// TwinCAT 3 PLC project plc_eta_factory_climate_room_automation
// ProgramVersion: 3.1.4024.12
// libraries:
//   AutomationBaseClasses, * (PTW TU Darmstadt)
//   Tc2_ControllerToolbox, * (Beckhoff Automation GmbH)
//   Tc2_MBus, * (Beckhoff Automation GmbH)
//   Tc2_Standard, * (Beckhoff Automation GmbH)
//   Tc2_System, * (Beckhoff Automation GmbH)
//   Tc2_Utilities, * (Beckhoff Automation GmbH)
//   Tc3_Module, * (Beckhoff Automation GmbH)
// project tree:
//   DUTs/04 Systems/ E_ActiveWallModulesControlMode.TcDUT, E_AirHandlingUnitControlMode.TcDUT, ST_ActiveWallModulesDefaultParameters.TcDUT, ST_ActiveWallModulesSetParameters.TcDUT, ST_AirHandlingUnitDefaultParameters.TcDUT, ST_PowerControlledHeaterState.TcDUT, ST_PowerControlledHeaterDefaultParameters.TcDUT, ST_AirHandlingUnitSetParameters.TcDUT, ST_AmbientState.TcDUT, ST_BufferStorageState.TcDUT
//   GVLs/ GlobalVariables.TcGVL, MBus.TcGVL
//   / MBusTask.TcTTO, PlcTask.TcTTO
//   POUs/01 Actuators/ FB_AirHandlingUnit.TcPOU, FB_PowerControlledHeaterThyristor.TcPOU, FB_PowerControlledHeaterFan.TcPOU, FB_PowerControlledHeaterContactor.TcPOU
//   POUs/02 Sensors/ FB_CO2Sensor.TcPOU, FB_HumiditySensor.TcPOU, FB_TemperatureSensor.TcPOU, FB_TemperatureSensorPCH.TcPOU, FB_JanitzaSensor.TcPOU
//   POUs/04 Systems/ FB_ActiveWallModulesSystem.TcPOU, FB_AirHandlingUnitSystem.TcPOU, FB_Ambient.TcPOU, FB_BufferStorage.TcPOU, FB_CNSystem.TcPOU, FB_HNLTSystem.TcPOU, FB_PowerControlledHeaterSystem.TcPOU
//   POUs/ MAIN.TcPOU, MBus_Communication.TcPOU

CONFIGURATION plc_eta_factory_climate_room_automation
    RESOURCE PLC ON TwinCAT3
        TASK MBusTask(INTERVAL := T#10ms, PRIORITY := 1);
        TASK PlcTask(INTERVAL := T#10ms, PRIORITY := 20);
        PROGRAM MBus_Communication WITH MBusTask : MBus_Communication;
        PROGRAM MAIN WITH PlcTask : MAIN;
    END_RESOURCE
END_CONFIGURATION

// ---- DUTs/04 Systems/E_ActiveWallModulesControlMode.TcDUT
{attribute 'qualified_only'}
{attribute 'strict'}
TYPE E_ActiveWallModulesControlMode :
(
	On := 0, //100% on
	Discrete := 1, //use hysteresis controller
	Continous := 2 //use PI-Controller
);
END_TYPE

// ---- DUTs/04 Systems/E_AirHandlingUnitControlMode.TcDUT
{attribute 'qualified_only'}
{attribute 'strict'}
TYPE E_AirHandlingUnitControlMode :
(
	On := 0, //100% on
	Discrete := 1, //use hysteresis controller
	Continous := 2 //use PI-Controller
);
END_TYPE

// ---- DUTs/04 Systems/ST_ActiveWallModulesDefaultParameters.TcDUT
TYPE ST_ActiveWallModulesDefaultParameters :
STRUCT
	aSetPointLimitsTemperature : ARRAY[1..2] OF REAL := [5,30];
END_STRUCT
END_TYPE

// ---- DUTs/04 Systems/ST_ActiveWallModulesSetParameters.TcDUT
{attribute 'OPC.UA.DA.StructuredType' := '1'}
TYPE ST_ActiveWallModulesSetParameters :
STRUCT
	bHeatingModeAlgorithm : BOOL;
	bHeatingModeManual : BOOL;
	nControlModeAlgorithm : E_ActiveWallModulesControlMode;
	nControlModeManual : E_ActiveWallModulesControlMode;
	fHysteresisRangeAlgorithm : REAL;
	fHysteresisRangeManual : REAL; 
END_STRUCT
END_TYPE

// ---- DUTs/04 Systems/ST_AirHandlingUnitDefaultParameters.TcDUT
TYPE ST_AirHandlingUnitDefaultParameters :
STRUCT
	aSetPointLimitsTemperature : ARRAY[1..2] OF REAL := [5,100];
END_STRUCT
END_TYPE

// ---- DUTs/04 Systems/ST_PowerControlledHeaterState.TcDUT
{attribute 'OPC.UA.DA.StructuredType' := '1'}
TYPE ST_PowerControlledHeaterState :
STRUCT
	fPowerTotal : REAL;
	sPowerUnit : STRING := 'W';
END_STRUCT
END_TYPE

// ---- DUTs/04 Systems/ST_PowerControlledHeaterDefaultParameters.TcDUT
TYPE ST_PowerControlledHeaterDefaultParameters :
STRUCT
	aSetPointLimitsPower : ARRAY[1..2] OF REAL := [0, 8000];
END_STRUCT
END_TYPE

// ---- DUTs/04 Systems/ST_AirHandlingUnitSetParameters.TcDUT
{attribute 'OPC.UA.DA.StructuredType' := '1'}
TYPE ST_AirHandlingUnitSetParameters :
STRUCT
	bHeatingModeAlgorithm : BOOL;
	bHeatingModeManual : BOOL;
	nControlModeAlgorithm : E_AirHandlingUnitControlMode;
	nControlModeManual : E_AirHandlingUnitControlMode;
	fHysteresisRangeAlgorithm : REAL;
	fHysteresisRangeManual : REAL;
END_STRUCT
END_TYPE

// ---- DUTs/04 Systems/ST_AmbientState.TcDUT
{attribute 'OPC.UA.DA.StructuredType' := '1'}
TYPE ST_AmbientState :
STRUCT
	fRoomTemperature : REAL;
	fRoomTemperatureUpperNO : REAL;
	fRoomTemperatureLowerNO : REAL;
	fRoomTemperatureUpperSO : REAL;
	fRoomTemperatureLowerSO : REAL;
	fRoomTemperatureUpperSW : REAL;
	fRoomTemperatureLowerSW : REAL;
	fRoomTemperatureUpperNW : REAL;
	fRoomTemperatureLowerNW : REAL;
	fOutsideTemperature : REAL;
	fOutsideTemperatureNorth : REAL;
	fOutsideTemperatureSouth : REAL;
	fOutsideTemperatureWest : REAL;
	fInletAHUTemperature : REAL;
	fOutletAHUTemperature : REAL;
	fInletVentilationTemperature : REAL;
	fOutletVentilationTemperature : REAL;
	sTemperatureUnit : STRING := 'degreeC';
	fRelativeHumidity : REAL;
	sRelativeHumidity : STRING := 'percent';
	fRoomCO2 : REAL;
	sRoomCO2 : STRING := 'ppm';
END_STRUCT
END_TYPE

// ---- DUTs/04 Systems/ST_BufferStorageState.TcDUT
{attribute 'OPC.UA.DA.StructuredType' := '1'}
TYPE ST_BufferStorageState :
STRUCT
	fUpperTemperature : REAL;
	fLowerTemperature : REAL;
	sTemperatureUnit : STRING := 'degreeC';
END_STRUCT
END_TYPE

// ---- GVLs/GlobalVariables.TcGVL
{attribute 'qualified_only'}
VAR_GLOBAL
	//cycle times
	tTaskCycleTime_MAIN				: TIME := T#10MS;
	tCtrlCycleTime_MAIN				: TIME := T#5S;
END_VAR

// ---- GVLs/MBus.TcGVL
{attribute 'qualified_only'}
VAR_GLOBAL
	IN_Zaehler AT %I* 		: ST_KL6781inData22B;
	OUT_Zaehler AT %Q* 		: ST_KL6781outData22B;
	Communication_MBus		: ST_MBUS_Communication;
	
	Telegramm_WMZ_196		: ARRAY[1..cMBUS_MaxTelegrams] OF ST_MBus_Data2;
	Telegramm_WMZ_193		: ARRAY[1..cMBUS_MaxTelegrams] OF ST_MBus_Data2;
	Telegramm_WMZ_491		: ARRAY[1..cMBUS_MaxTelegrams] OF ST_MBus_Data2;
	Telegramm_WMZ_493		: ARRAY[1..cMBUS_MaxTelegrams] OF ST_MBus_Data2;
	Telegramm_WMZ_393		: ARRAY[1..cMBUS_MaxTelegrams] OF ST_MBus_Data2;
	Telegramm_WMZ_198		: ARRAY[1..cMBUS_MaxTelegrams] OF ST_MBus_Data2;
	Telegramm_WMZ_246		: ARRAY[1..cMBUS_MaxTelegrams] OF ST_MBus_Data2;
	Telegramm_WMZ_247		: ARRAY[1..cMBUS_MaxTelegrams] OF ST_MBus_Data2;
	Telegramm_WMZ_592		: ARRAY[1..cMBUS_MaxTelegrams] OF ST_MBus_Data2;
END_VAR

// ---- POUs/MBus_Communication.TcPOU
PROGRAM MBus_Communication
VAR
	Communication_Terminal	: FB_MBUSKL6781;
	
	WMZ_196					: FB_MBUS_General_Ext;
	WMZ_193					: FB_MBUS_General_Ext;
	WMZ_491					: FB_MBUS_General_Ext;
	WMZ_493					: FB_MBUS_General_Ext;
	WMZ_393					: FB_MBUS_General_Ext;
	WMZ_198					: FB_MBUS_General_Ext;
	WMZ_246					: FB_MBUS_General_Ext;
	WMZ_247					: FB_MBUS_General_Ext;
	WMZ_592					: FB_MBUS_General_Ext;
	
	//define secondary addresses
	adrWMZ_196			: ST_MBUS_SecAdr := (udiIdNumber:=16#91453216);
	adrWMZ_193			: ST_MBUS_SecAdr := (udiIdNumber:=16#91057344);
	adrWMZ_491			: ST_MBUS_SecAdr := (udiIdNumber:=16#91057337);
	adrWMZ_493			: ST_MBUS_SecAdr := (udiIdNumber:=16#85052762);
	adrWMZ_393			: ST_MBUS_SecAdr := (udiIdNumber:=16#93556978);
	adrWMZ_198			: ST_MBUS_SecAdr := (udiIdNumber:=16#72888375);
	adrWMZ_246			: ST_MBUS_SecAdr := (udiIdNumber:=16#72888412);
	adrWMZ_247			: ST_MBUS_SecAdr := (udiIdNumber:=16#72888417);
	adrWMZ_592			: ST_MBUS_SecAdr := (udiIdNumber:=16#30356999);
END_VAR

Communication_Terminal(stComIn := MBus.IN_Zaehler, stComOut := MBus.OUT_Zaehler, stCom := MBus.Communication_MBus);

WMZ_196(usiAddress := 253, stSecAdr := adrWMZ_196, stCom := MBus.Communication_MBus, arrTelegram => MBus.Telegramm_WMZ_196);
WMZ_193(usiAddress := 253, stSecAdr := adrWMZ_193, stCom := MBus.Communication_MBus, arrTelegram => MBus.Telegramm_WMZ_193);
WMZ_198(usiAddress := 253, stSecAdr := adrWMZ_198, stCom := MBus.Communication_MBus, arrTelegram => MBus.Telegramm_WMZ_198);

WMZ_246(usiAddress := 253, stSecAdr := adrWMZ_246, stCom := MBus.Communication_MBus, arrTelegram => MBus.Telegramm_WMZ_246);
WMZ_247(usiAddress := 253, stSecAdr := adrWMZ_247, stCom := MBus.Communication_MBus, arrTelegram => MBus.Telegramm_WMZ_247);

WMZ_393(usiAddress := 253, stSecAdr := adrWMZ_393, stCom := MBus.Communication_MBus, arrTelegram => MBus.Telegramm_WMZ_393);

WMZ_491(usiAddress := 253, stSecAdr := adrWMZ_491, stCom := MBus.Communication_MBus, arrTelegram => MBus.Telegramm_WMZ_491);
WMZ_493(usiAddress := 253, stSecAdr := adrWMZ_493, stCom := MBus.Communication_MBus, arrTelegram => MBus.Telegramm_WMZ_493);

WMZ_592(usiAddress := 253, stSecAdr := adrWMZ_592, stCom := MBus.Communication_MBus, arrTelegram => MBus.Telegramm_WMZ_592);

END_PROGRAM

// ---- POUs/MAIN.TcPOU
PROGRAM MAIN
VAR
	stRoomCheckDefaultParameters : ST_RangeCheckDefaultParameters := (tTaskCycleTime := GlobalVariables.tCtrlCycleTime_MAIN, tCtrlCycleTime := GlobalVariables.tCtrlCycleTime_MAIN, fRestoreDifference := 4);
	Room_Check : FB_RangeCheck := (ST_DefaultParameters := stRoomCheckDefaultParameters);
	
	Ambient : FB_Ambient;
	BufferStorage : FB_BufferStorage;
	ActiveWallModules : FB_ActiveWallModulesSystem;
	AirHandlingUnit : FB_AirHandlingUnitSystem;
	CN : FB_CNSystem;
	HNLT: FB_HNLTSystem;
	
	PCH : FB_PowerControlledHeaterSystem;
END_VAR

Ambient();
BufferStorage();

//set algorithm permission depending on production mode to control structs
Room_Check(fInput := Ambient.localState.fRoomTemperature,
	fLowerLimit := 5,
	fUpperLimit := 30);

ActiveWallModules(bSetStatusOnAutomatic := FALSE,
	fSetPointAutomatic := 0,
	bAlgorithmPermission := Room_Check.bPermission,
	bHeatingModeAutomatic := FALSE,
	fHysteresisRangeAutomatic := 3,
	stAmbientState := Ambient.localState);
	
AirHandlingUnit(bSetStatusOnAutomatic := FALSE,
	fSetPointAutomatic := 0,
	bAlgorithmPermission := Room_Check.bPermission,
	bHeatingModeAutomatic := FALSE,
	fHysteresisRangeAutomatic := 3,
	stAmbientState := Ambient.localState);
	
CN(bSetStatusOnAutomatic := FALSE,
	fSetPointAutomatic := 0,
	bAlgorithmPermission := Room_Check.bPermission);

HNLT();	
	
PCH(bSetStatusOnAutomatic := FALSE,
	bAlgorithmPermission := Room_Check.bPermission,
	fSetPointAutomatic := 0);

END_PROGRAM

// ---- POUs/04 Systems/FB_Ambient.TcPOU
FUNCTION_BLOCK FB_Ambient
VAR_INPUT
END_VAR
VAR_OUTPUT
	{attribute 'OPC.UA.DA' := '1'}
	localState : ST_AmbientState;
END_VAR
VAR
	//sensors
	UpperRoomTemperature_SW : FB_TemperatureSensor; //south west
	LowerRoomTemperature_SW : FB_TemperatureSensor;
	UpperRoomTemperature_NW : FB_TemperatureSensor; //north west
	LowerRoomTemperature_NW : FB_TemperatureSensor;
	UpperRoomTemperature_NO : FB_TemperatureSensor;//north east
	LowerRoomTemperature_NO : FB_TemperatureSensor;
	UpperRoomTemperature_SO : FB_TemperatureSensor; //south east
	LowerRoomTemperature_SO : FB_TemperatureSensor;
	
	OutsideTemperature_North : FB_TemperatureSensor;
	OutsideTemperature_South : FB_TemperatureSensor;
	OutsideTemperature_West : FB_TemperatureSensor;
	
	InletAHUTemperature : AutomationBaseClasses.FB_TemperatureSensor; //inlet temperature from climate room internal AHU (Air Handling Unit)
	OutletAHUTemperature : AutomationBaseClasses.FB_TemperatureSensor; //outlet temperature from climate room internal AHU
	
	InletVentilationTemperature : AutomationBaseClasses.FB_TemperatureSensor; //inlet temperature from building ventilation
	OutletVentilationTemperature : AutomationBaseClasses.FB_TemperatureSensor; //outlet temperature from building ventilation
	
	RoomHumidity : FB_HumiditySensor;
	RoomCO2 : FB_CO2Sensor;
END_VAR

UpperRoomTemperature_SW();
UpperRoomTemperature_SW.GetState_AI();
LowerRoomTemperature_SW();
LowerRoomTemperature_SW.GetState_AI();
UpperRoomTemperature_NW();
UpperRoomTemperature_NW.GetState_AI();
LowerRoomTemperature_NW();
LowerRoomTemperature_NW.GetState_AI();
UpperRoomTemperature_NO();
UpperRoomTemperature_NO.GetState_AI();
LowerRoomTemperature_NO();
LowerRoomTemperature_NO.GetState_AI();
UpperRoomTemperature_SO();
UpperRoomTemperature_SO.GetState_AI();
LowerRoomTemperature_SO();
LowerRoomTemperature_SO.GetState_AI();

OutsideTemperature_North();
OutsideTemperature_North.GetState_AI();
OutsideTemperature_South();
OutsideTemperature_South.GetState_AI();
OutsideTemperature_West();
OutsideTemperature_West.GetState_AI();

InletAHUTemperature();
InletAHUTemperature.GetState_AI();
OutletAHUTemperature();
OutletAHUTemperature.GetState_AI();
InletVentilationTemperature();
InletVentilationTemperature.GetState_AI();
OutletVentilationTemperature();
OutletVentilationTemperature.GetState_AI();

RoomHumidity();
RoomHumidity.GetState_AI();

RoomCO2();
RoomCO2.GetState_AI();

SetState();

METHOD PROTECTED SetState : BOOL
VAR_INPUT
END_VAR
localState.fRelativeHumidity := RoomHumidity.fHumidity;
localState.fRoomCO2 := RoomCO2.fCO2;

localState.fRoomTemperatureUpperNO := UpperRoomTemperature_NO.fTemperature;
localState.fRoomTemperatureLowerNO := LowerRoomTemperature_NO.fTemperature;
localState.fRoomTemperatureUpperSO := UpperRoomTemperature_SO.fTemperature;
localState.fRoomTemperatureLowerSO := LowerRoomTemperature_SO.fTemperature;
localState.fRoomTemperatureUpperSW := UpperRoomTemperature_SW.fTemperature;
localState.fRoomTemperatureLowerSW := LowerRoomTemperature_SW.fTemperature;
localState.fRoomTemperatureUpperNW := UpperRoomTemperature_NW.fTemperature;
localState.fRoomTemperatureLowerNW := LowerRoomTemperature_NW.fTemperature;

localState.fInletAHUTemperature := InletAHUTemperature.fTemperature;
localState.fOutletAHUTemperature := OutletAHUTemperature.fTemperature;
localState.fInletVentilationTemperature := InletVentilationTemperature.fTemperature;
localState.fOutletVentilationTemperature := OutletVentilationTemperature.fTemperature;

//room temperature is currently calclated as mean value from all room values
localState.fRoomTemperature := (localState.fRoomTemperatureUpperNO+localState.fRoomTemperatureLowerNO+localState.fRoomTemperatureUpperSO+localState.fRoomTemperatureLowerSO+localState.fRoomTemperatureUpperSW+localState.fRoomTemperatureLowerSW+localState.fRoomTemperatureUpperNW+localState.fRoomTemperatureLowerNW)/8;

localState.fOutsideTemperatureNorth := OutsideTemperature_North.fTemperature;
localState.fOutsideTemperatureSouth := OutsideTemperature_South.fTemperature;
localState.fOutsideTemperatureWest := OutsideTemperature_West.fTemperature;

//outside temperature is currently calclated as mean value from all outside values
localState.fOutsideTemperature := (localState.fOutsideTemperatureNorth+localState.fOutsideTemperatureSouth+localState.fOutsideTemperatureWest)/3;
END_METHOD

END_FUNCTION_BLOCK

// ---- POUs/02 Sensors/FB_TemperatureSensor.TcPOU
FUNCTION_BLOCK FB_TemperatureSensor EXTENDS FB_Sensor
VAR_INPUT
END_VAR
VAR_OUTPUT
	fTemperature : REAL; //measured temperature in °C
END_VAR
VAR
	//I/O-Links
	temperature_IN AT %I* : INT;
	
END_VAR

METHOD GetState_AI : BOOL
VAR_INPUT
END_VAR
fTemperature := (temperature_IN / 32767.0)*50.0;  //conversion: scaled to temperature 0-50 °C from 0 - 10 V

//sensor state
sensorState.fValue := fTemperature;
sensorState.sUnit := 'degreeC';
END_METHOD

END_FUNCTION_BLOCK

// ---- POUs/02 Sensors/FB_HumiditySensor.TcPOU
FUNCTION_BLOCK FB_HumiditySensor EXTENDS FB_Sensor
VAR_INPUT
END_VAR
VAR_OUTPUT
	fHumidity : REAL; //measured relative humidity
END_VAR
VAR
	//I/O-Links
	humidity_IN AT %I* : INT;
	
END_VAR

METHOD GetState_AI : BOOL
VAR_INPUT
END_VAR
//Humidity := (humidity_IN / 32767.0)- Offset 10% ;
fHumidity := (humidity_IN / 32767.0)-0.1;

(*Umrechnungsfaktor muss noch angepasst werden
0 ist minimaler Wert	:= 0 V -> 0 % Luftfeuchtigkeit
32767 ist maximaler Wert := 10 V -> 100 % Luftfeuchtigkeit
*)

//sensor state
sensorState.fValue := fHumidity;
sensorState.sUnit := 'percent';
END_METHOD

END_FUNCTION_BLOCK

// ---- POUs/02 Sensors/FB_CO2Sensor.TcPOU
FUNCTION_BLOCK FB_CO2Sensor EXTENDS FB_Sensor
VAR_INPUT
END_VAR
VAR_OUTPUT
	fCO2 : REAL; //measured CO2 concentration in ppm
END_VAR
VAR
	//I/O-Links
	CO2_IN AT %I* : INT;
	
END_VAR

METHOD GetState_AI : BOOL
VAR_INPUT
END_VAR
fCO2 :=  (CO2_IN / 32767.0)*2000; //conversion

//sensor state
sensorState.fValue := fCO2;
sensorState.sUnit := 'ppm';
END_METHOD

END_FUNCTION_BLOCK

// ---- POUs/04 Systems/FB_BufferStorage.TcPOU
FUNCTION_BLOCK FB_BufferStorage
VAR_INPUT
END_VAR
VAR_OUTPUT
	{attribute 'OPC.UA.DA' := '1'}
	localState : ST_BufferStorageState;
END_VAR
VAR
	//sensors
	UpperBufferTemperature : AutomationBaseClasses.FB_TemperatureSensor;
	LowerBufferTemperature : AutomationBaseClasses.FB_TemperatureSensor;
	
	WMZ198 : FB_MollineC3HeatCounter;
	
END_VAR

UpperBufferTemperature();
UpperBufferTemperature.GetState_AI();

LowerBufferTemperature();
LowerBufferTemperature.GetState_AI();

WMZ198(aHeatCounterTelegramm := MBus.Telegramm_WMZ_198);

SetState();

METHOD PROTECTED SetState : BOOL
VAR_INPUT
END_VAR
localState.fUpperTemperature := UpperBufferTemperature.fTemperature;
localState.fLowerTemperature := LowerBufferTemperature.fTemperature;
END_METHOD

END_FUNCTION_BLOCK

// ---- POUs/04 Systems/FB_ActiveWallModulesSystem.TcPOU
FUNCTION_BLOCK FB_ActiveWallModulesSystem EXTENDS FB_SystemContinous
VAR_INPUT
	nControlModeAutomatic : E_ActiveWallModulesControlMode;	
	bHeatingModeAutomatic : BOOL; //control mode: 0 = heating mode; 1 = cooling mode
	fHysteresisRangeAutomatic : REAL; //default unequalt to zero
	stAmbientState : ST_AmbientState;
END_VAR
VAR_OUTPUT
END_VAR
VAR
	{attribute 'OPC.UA.DA' := '1'}
 	localSetParameters : ST_ActiveWallModulesSetParameters;
	
	localDefaultParameters : ST_ActiveWallModulesDefaultParameters;
	
	//pumps
	stPU492DefaultParameters : ST_PumpGrundfosMagna3DefaultParameters;
	stPU592DefaultParameters : ST_PumpGrundfosMagna3DefaultParameters;
	PU492 : FB_PumpGrundfosMagna3 := (ST_DefaultParameters := stPU492DefaultParameters);
	PU592 : FB_PumpGrundfosMagna3 := (ST_DefaultParameters := stPU592DefaultParameters);	
	//valves
	stSV490DefaultParameters : ST_DiscreteValveDefaultParameters;
	stSV491DefaultParameters : ST_DiscreteValveDefaultParameters;
	stSV493DefaultParameters : ST_DiscreteValveDefaultParameters;
	stSV494DefaultParameters : ST_DiscreteValveDefaultParameters;
	
	//fDefaultPosition = 100 means bypass for bSetStatusOn = false
	stRV492DefaultParameters : ST_MixingValveDefaultParameters := (bFeedbackSignal := FALSE, fControllerAmplification := 5, tControllerIntegralTime := T#100M, bARWOnIPartOnly := FALSE, fDefaultPosition := 100, tTaskCycleTime := GlobalVariables.tTaskCycleTime_MAIN, tCtrlCycleTime := GlobalVariables.tCtrlCycleTime_MAIN);
	
	SV490 : FB_DiscreteValve := (ST_DefaultParameters := stSV490DefaultParameters);
	SV491 : FB_DiscreteValve := (ST_DefaultParameters := stSV491DefaultParameters);
	SV493 : FB_DiscreteValve := (ST_DefaultParameters := stSV493DefaultParameters);
	SV494 : FB_DiscreteValve := (ST_DefaultParameters := stSV494DefaultParameters);
	
	RV492 : FB_MixingValve := (ST_DefaultParameters := stRV492DefaultParameters); 
	
	//sensors
	TVL492 : AutomationBaseClasses.FB_TemperatureSensor; //supply temperature
	TRL492 : AutomationBaseClasses.FB_TemperatureSensor; //return temperature
	TVL592 : AutomationBaseClasses.FB_TemperatureSensor; //supply temperature walls
	TRL592 : AutomationBaseClasses.FB_TemperatureSensor; //return temperature walls
	
	WMZ491 : FB_MollineC3HeatCounter; //cooling network
	WMZ493 : FB_MollineC3HeatCounter; //heating network
	WMZ592 : FB_MollineC3HeatCounter;
	
	//internal variables
	bHeatingMode 			: BOOL;
	bSetStatusOn_PU492 		: BOOL;
	bSetStatusOn_PU592 		: BOOL;
	bSetStatusOn_SV490		: BOOL;
	bSetStatusOn_SV491		: BOOL;
	bSetStatusOn_SV493		: BOOL;
	bSetStatusOn_SV494		: BOOL;
	bSetStatusOn_RV492		: BOOL;
	
	nControlMode_RV492 		: E_MixingValveControlMode;
	fSetPoint_RV492 		: REAL;	
	nControlMode			: E_ActiveWallModulesControlMode;
	fHysteresisRange		: REAL;

	//controller
	PI_Controller				: FB_CTRL_PI;
	PI_Controller_Parameters	: ST_CTRL_PI_PARAMS;
	TwoPointControllerHeating		: FB_CTRL_2POINT;
	TwoPointControllerCooling		: FB_CTRL_2POINT;
	TwoPointControllerParameters 	: ST_CTRL_2POINT_PARAMS;
	
	//triggers
	SwitchToHeating : R_TRIG;
	SwitchToCooling : F_TRIG;
	bFinishedSwitchMode : BOOL := TRUE;

	
	//clock
	bStartTimer : BOOL;
	Timer : TON;

END_VAR

SelectLocalControlMode();
SwitchToHeating(CLK := bHeatingMode);
SwitchToCooling(CLK := bHeatingMode);

Timer(IN := bStartTimer,
	PT := T#120S);
MAIN();

//pumps
PU492.GetState_Profibus();
PU492(bSetStatusOnAutomatic := bSetStatusOn_PU492,
	bAlgorithmPermission := bAlgorithmPermission,
	fSetPointAutomatic := 100,
	nControlModeAutomatic := 0);
PU492.SetState_Profibus();

PU592.GetState_Profibus();
PU592(bSetStatusOnAutomatic := bSetStatusOn_PU592,
	bAlgorithmPermission := bAlgorithmPermission,
	fSetPointAutomatic := 100,
	nControlModeAutomatic := 0);
PU592.SetState_Profibus();

//valves
RV492.GetState_AI();
RV492(bSetStatusOnAutomatic := bSetStatusOn_RV492,
	fSetPointAutomatic := fSetPoint_RV492,
	nControlModeAutomatic := nControlMode_RV492,
	bAlgorithmPermission := bAlgorithmPermission,
	fTemperatureExternal := stAmbientState.fRoomTemperature);
RV492.SetState_AO();

SV490.GetState_BI();
SV490(bSetStatusOnAutomatic := bSetStatusOn_SV490,
	bAlgorithmPermission := bAlgorithmPermission);
SV490.SetState_BO();

SV491.GetState_BI();
SV491(bSetStatusOnAutomatic := bSetStatusOn_SV491,
	bAlgorithmPermission := bAlgorithmPermission);
SV491.SetState_BO();

SV493.GetState_BI();
SV493(bSetStatusOnAutomatic := bSetStatusOn_SV493,
	bAlgorithmPermission := bAlgorithmPermission);
SV493.SetState_BO();

SV494.GetState_BI();
SV494(bSetStatusOnAutomatic := bSetStatusOn_SV494,
	bAlgorithmPermission := bAlgorithmPermission);
SV494.SetState_BO();

//sensors
TVL492();
TVL492.GetState_AI();
TRL492();
TRL492.GetState_AI();

TVL592();
TVL592.GetState_AI();
TRL592();
TRL592.GetState_AI();

WMZ491(aHeatCounterTelegramm := MBus.Telegramm_WMZ_491);
WMZ493(aHeatCounterTelegramm := MBus.Telegramm_WMZ_493);
WMZ592(aHeatCounterTelegramm := MBus.Telegramm_WMZ_592);

METHOD PROTECTED  CheckError : BOOL
VAR_INPUT
END_VAR
VAR_OUTPUT
	bError : BOOL;
END_VAR
VAR
	bError_PU492 : BOOL;
	bError_PU592 : BOOL;
END_VAR
//check pumps for errors
bError_PU492 := PU492.bError;
bError_PU592 := PU592.bError;

bError := bError_PU492 OR bError_PU592;
END_METHOD

METHOD PRIVATE LocalControl : BOOL
VAR_INPUT
END_VAR

VAR
	TwoPointControllerOutput : BOOL;
END_VAR
CASE nControlMode OF
	0: //100%
	nControlMode_RV492 := 0;	//position mode
	fSetPoint_RV492 := 0; //0 is fully opened
	
	1: //Hysteresis
	nControlMode_RV492 := 0;	//position mode
	TwoPointControllerParameters.tCtrlCycleTime := T#1S;
	TwoPointControllerParameters.tTaskCycleTime := T#10MS;
	IF fHysteresisRange < 1 THEN
		TwoPointControllerParameters.fHysteresisRange := 1;
	ELSE
		TwoPointControllerParameters.fHysteresisRange := fHysteresisRange;
	END_IF;
	
	TwoPointControllerHeating(
			fSetpointValue := fSetPoint,
			fActualValue := stAmbientState.fRoomTemperature,
			bManSyncValue := 0,
			bSync := FALSE,
			emode := 2,
			stParams := TwoPointControllerParameters);
			
	TwoPointControllerCooling(
			fSetpointValue := stAmbientState.fRoomTemperature,
			fActualValue := fSetPoint,
			bManSyncValue := 0,
			bSync := FALSE,
			emode := 2,
			stParams := TwoPointControllerParameters);

	
	IF bHeatingMode THEN
		TwoPointControllerOutput := TwoPointControllerHeating.bOut;
	ELSE
		TwoPointControllerOutput := TwoPointControllerCooling.bOut;
	END_IF
	
	IF TwoPointControllerOutput THEN
		bSetStatusOn_PU492 := TRUE;
		bSetStatusOn_PU592 := TRUE;
		bSetStatusOn_RV492 := TRUE;
		fSetPoint_RV492 := 0; //0 is fully opened
	ELSE
		bSetStatusOn_PU492 := FALSE;
		bSetStatusOn_PU592 := FALSE;
		bSetStatusOn_RV492 := FALSE;
		fSetPoint_RV492 := 100; //0 is fully opened
	END_IF	
	
			
	2: //Continous with PI-Controller
	IF bHeatingMode THEN
		nControlMode_RV492 := 2; //inverted because of internal valve control mode
	ELSE
		nControlMode_RV492 := 1;
	END_IF
	fSetPoint_RV492 := fSetPoint;
	bSetStatusOn_PU492 := TRUE;
	bSetStatusOn_PU592 := TRUE;

END_CASE
END_METHOD

METHOD PROTECTED  Operational : BOOL
VAR_INPUT
END_VAR
VAR_OUTPUT
	bSwitchToWorking : BOOL := FALSE;
END_VAR
bSetStatusOn_RV492 := TRUE;

bSetStatusOn_PU492 := TRUE;
bSetStatusOn_PU592 := TRUE;

IF PU492.bStatusOn AND PU592.bStatusOn THEN
	bSwitchToWorking := TRUE;
END_IF
END_METHOD

METHOD PROTECTED  RampDown : BOOL
VAR_INPUT
END_VAR
VAR_OUTPUT
	bRampDownFinished : BOOL := FALSE;
END_VAR
bSetStatusOn_PU492 := FALSE;
bSetStatusOn_PU592 := FALSE;

IF NOT PU492.bStatusOn AND NOT PU592.bStatusOn THEN
	bSetStatusOn_RV492 := FALSE;
	
	bSetStatusOn_SV493 := FALSE;
	bSetStatusOn_SV494 := FALSE;
	
	bSetStatusOn_SV490 := FALSE;
	bSetStatusOn_SV491 := FALSE;
	bStartTimer := TRUE;
	IF Timer.Q THEN
		bRampDownFinished := TRUE;
		bStartTimer := FALSE;
	END_IF
END_IF
END_METHOD

METHOD PROTECTED  RampUp : BOOL
VAR_INPUT
END_VAR
VAR_OUTPUT
	bRampUpFinished : BOOL := FALSE;
END_VAR
bSetStatusOn_RV492 := TRUE;
IF bHeatingMode THEN
	bSetStatusOn_SV493 := TRUE;
	bSetStatusOn_SV494 := TRUE;
	
	bSetStatusOn_SV490 := FALSE;
	bSetStatusOn_SV491 := FALSE;
	
	nControlMode_RV492 := 1; //heating mode
ELSE
	bSetStatusOn_SV493 := FALSE;
	bSetStatusOn_SV494 := FALSE;
	
	bSetStatusOn_SV490 := TRUE;
	bSetStatusOn_SV491 := TRUE;
	
	nControlMode_RV492 := 2; //cooling mode
END_IF

bStartTimer := TRUE;
IF Timer.Q THEN
	bStartTimer := FALSE;
	bRampUpFinished := TRUE;
END_IF
END_METHOD

METHOD PRIVATE SelectLocalControlMode : BOOL
VAR_INPUT
END_VAR
VAR
END_VAR
IF control.bManualModeActivated THEN
	bHeatingMode := localSetParameters.bHeatingModeManual;
	nControlMode := localSetParameters.nControlModeManual;
	fHysteresisRange := localSetParameters.fHysteresisRangeManual;
ELSIF control.bAlgorithmModeActivated AND bAlgorithmPermission THEN
	bHeatingMode := localSetParameters.bHeatingModeAlgorithm;
	nControlMode := localSetParameters.nControlModeAlgorithm;
	fHysteresisRange := localSetParameters.fHysteresisRangeAlgorithm;
ELSE
	bHeatingMode := bHeatingModeAutomatic;
	nControlMode := nControlModeAutomatic;
	fHysteresisRange := fHysteresisRangeAutomatic;
END_IF
END_METHOD

METHOD PROTECTED   SetSetPointLimits : BOOL
VAR_INPUT
END_VAR
VAR_OUTPUT
END_VAR
aSetPointLimits[1] := localDefaultParameters.aSetPointLimitsTemperature[1];
aSetPointLimits[2] := localDefaultParameters.aSetPointLimitsTemperature[2];
END_METHOD

METHOD PROTECTED  SetState : BOOL
VAR_INPUT
END_VAR
VAR_OUTPUT
END_VAR
fOperatingPoint := stAmbientState.fRoomTemperature;

controlState.bStatusOn := bSetStatusOn;
setPointState.aSetPointLimits := aSetPointLimits;
setPointState.fSetPoint := fSetPoint;
setPointState.fOperatingPoint := fOperatingPoint;
setPointState.sSetPointUnit := 'degreeC';
setPointState.sOperatingPointUnit := 'degreeC';
END_METHOD

METHOD PRIVATE SwitchMode : BOOL
VAR_INPUT
	bSwitchToHeating : BOOL; //if false switch to cooling
END_VAR
VAR_OUTPUT
	bFinishedSwitchMode : BOOL;
END_VAR
VAR_INST
	bRampDownFinished : BOOL := FALSE;
END_VAR
IF bSwitchToHeating THEN
	//turn off pumps first		
	bSetStatusOn_PU492 := FALSE;
	bSetStatusOn_PU592 := FALSE;
	
	//SV can switch simultanously
	bSetStatusOn_SV490 := FALSE;
	bSetStatusOn_SV491 := FALSE;
	
	bSetStatusOn_SV493 := TRUE;
	bSetStatusOn_SV494 := TRUE;
	bFinishedSwitchMode := FALSE;
	bStartTimer := TRUE;
	IF Timer.Q THEN
		bStartTimer := FALSE;
		bRampDownFinished := TRUE;
		bFinishedSwitchMode := TRUE;
		bSetStatusOn_PU492 := TRUE;
		bSetStatusOn_PU592 := TRUE;
	END_IF
ELSE
	//turn off pumps first		
	bSetStatusOn_PU492 := FALSE;
	bSetStatusOn_PU592 := FALSE;

	//SV can switch simultanously
	bSetStatusOn_SV490 := TRUE;
	bSetStatusOn_SV491 := TRUE;
	
	bSetStatusOn_SV493 := FALSE;
	bSetStatusOn_SV494 := FALSE;
	bFinishedSwitchMode := FALSE;
	bStartTimer := TRUE;
	IF Timer.Q THEN
		bStartTimer := FALSE;
		bRampDownFinished := TRUE;
		bFinishedSwitchMode := TRUE;
		bSetStatusOn_PU492 := TRUE;
		bSetStatusOn_PU592 := TRUE;
	END_IF
END_IF
END_METHOD

METHOD PROTECTED  Working : BOOL
VAR_INPUT
END_VAR
VAR_OUTPUT
	bSwitchToOperational : BOOL := FALSE;
END_VAR
LocalControl();

IF ((SwitchToHeating.Q OR SwitchToCooling.Q) OR NOT bFinishedSwitchMode) THEN
	
	SwitchMode(bSwitchToHeating := bHeatingMode,
		bFinishedSwitchMode => bFinishedSwitchMode);
END_IF;
END_METHOD

END_FUNCTION_BLOCK

// ---- POUs/04 Systems/FB_AirHandlingUnitSystem.TcPOU
FUNCTION_BLOCK FB_AirHandlingUnitSystem EXTENDS FB_SystemContinous
VAR_INPUT
	nControlModeAutomatic : E_AirHandlingUnitControlMode;
	bHeatingModeAutomatic : BOOL; //control mode: 0 = heating mode; 1 = cooling mode
	fHysteresisRangeAutomatic : REAL; //default unequalt to zero	
	stAmbientState : ST_AmbientState;
END_VAR
VAR_OUTPUT
END_VAR
VAR
	{attribute 'OPC.UA.DA' := '1'}
 	localSetParameters : ST_AirHandlingUnitSetParameters;
	
	localDefaultParameters : ST_AirHandlingUnitDefaultParameters;
	
	//AHU
	AHU : FB_AirHandlingUnit;
	
	//pumps
	stPU193DefaultParameters : ST_PumpGrundfosMagna3DefaultParameters;
	stPU393DefaultParameters : ST_PumpGrundfosMagna3DefaultParameters;
	PU193 : FB_PumpGrundfosMagna3 := (ST_DefaultParameters := stPU193DefaultParameters);
	PU393 : FB_PumpGrundfosMagna3 := (ST_DefaultParameters := stPU393DefaultParameters);

	//valves
	stRV193DefaultParameters : ST_MixingValveDefaultParameters := (bFeedbackSignal := FALSE, fControllerAmplification := 5, tControllerIntegralTime := T#100M, bARWOnIPartOnly := FALSE, tTaskCycleTime := GlobalVariables.tTaskCycleTime_MAIN, tCtrlCycleTime := GlobalVariables.tCtrlCycleTime_MAIN);
	stRV393DefaultParameters : ST_MixingValveDefaultParameters := (bFeedbackSignal := FALSE, fControllerAmplification := 5, tControllerIntegralTime := T#100M, bARWOnIPartOnly := FALSE, tTaskCycleTime := GlobalVariables.tTaskCycleTime_MAIN, tCtrlCycleTime := GlobalVariables.tCtrlCycleTime_MAIN);
	
	RV193 : FB_MixingValve := (ST_DefaultParameters := stRV193DefaultParameters);
	RV393 : FB_MixingValve := (ST_DefaultParameters := stRV393DefaultParameters);	
	
	//sensors
	TVL193 : AutomationBaseClasses.FB_TemperatureSensor; //supply temperature cooling
	TRL193 : AutomationBaseClasses.FB_TemperatureSensor; //return temperature cooling
	TVL393 : AutomationBaseClasses.FB_TemperatureSensor; //supply temperature heating
	TRL393 : AutomationBaseClasses.FB_TemperatureSensor; //return temperature heating
	
	WMZ193 : FB_MollineC3HeatCounter; //cooling network
	WMZ393 : FB_MollineC3HeatCounter; //heating network
	
	//internal variables
	bHeatingMode 			: BOOL;

	bSetStatusOn_AHU		: BOOL;
	bSetStatusOn_PU193 		: BOOL;
	bSetStatusOn_PU393 		: BOOL;
	bSetStatusOn_RV193		: BOOL;
	bSetStatusOn_RV393		: BOOL;
	
	//local control	
	nControlMode			: E_AirHandlingUnitControlMode;
	
	nControlMode_RV193 		: E_MixingValveControlMode;	
	nControlMode_RV393 		: E_MixingValveControlMode;
	nControlMode_PU193		: AutomationBaseClasses.E_GrundfosMagna3ControlMode;
	nControlMode_PU393		: AutomationBaseClasses.E_GrundfosMagna3ControlMode;
	fSetPoint_RV193 		: REAL;
	fSetPoint_RV393 		: REAL;
	fHysteresisRange		: REAL;
	
	TwoPointControllerHeating		: FB_CTRL_2POINT;
	TwoPointControllerCooling		: FB_CTRL_2POINT;
	TwoPointControllerParameters 	: ST_CTRL_2POINT_PARAMS;
	
	//triggers
	SwitchToHeating : R_TRIG;
	SwitchToCooling : F_TRIG;
	bFinishedSwitchMode : BOOL := TRUE;
	
	//clock
	bStartTimer : BOOL;
	Timer : TON;

	
END_VAR

SelectLocalControlMode();
SwitchToHeating(CLK := bHeatingMode);
SwitchToCooling(CLK := bHeatingMode);

Timer(IN := bStartTimer,
	PT := T#120S);
MAIN();

AHU.GetState();
AHU(fSetPointAutomatic :=  100,
	bSetStatusOnAutomatic := bSetStatusOn_AHU,
	bAlgorithmPermission := bAlgorithmPermission);
AHU.SetState();

//pumps
PU193.GetState_Profibus();
PU193(bSetStatusOnAutomatic := bSetStatusOn_PU193,
	bAlgorithmPermission := bAlgorithmPermission,
	fSetPointAutomatic := 100,
	nControlModeAutomatic := nControlMode_PU193);
PU193.SetState_Profibus();

PU393.GetState_Profibus();
PU393(bSetStatusOnAutomatic := bSetStatusOn_PU393,
	bAlgorithmPermission := bAlgorithmPermission,
	fSetPointAutomatic := 100,
	nControlModeAutomatic := nControlMode_PU393);
PU393.SetState_Profibus();


//valves
RV193.GetState_AI();
RV193(bSetStatusOnAutomatic := bSetStatusOn_RV193,
	fSetPointAutomatic := fSetPoint_RV193,
	nControlModeAutomatic := nControlMode_RV193,
	bAlgorithmPermission := bAlgorithmPermission,
	fTemperatureExternal := stAmbientState.fRoomTemperature);
RV193.SetState_AO();

RV393.GetState_AI();
RV393(bSetStatusOnAutomatic := bSetStatusOn_RV393,
	fSetPointAutomatic := fSetPoint_RV393,
	nControlModeAutomatic := nControlMode_RV393,
	bAlgorithmPermission := bAlgorithmPermission,
	fTemperatureExternal := stAmbientState.fRoomTemperature);
RV393.SetState_AO();

//sensors
TVL193();
TVL193.GetState_AI();
TRL193();
TRL193.GetState_AI();

TVL393();
TVL393.GetState_AI();
TRL393();
TRL393.GetState_AI();

WMZ193(aHeatCounterTelegramm := MBus.Telegramm_WMZ_193);
WMZ393(aHeatCounterTelegramm := MBus.Telegramm_WMZ_393);

METHOD PROTECTED  CheckError : BOOL
VAR_INPUT
END_VAR
VAR_OUTPUT
	bError : BOOL;
END_VAR
VAR
	bError_PU193 : BOOL;
	bError_PU393 : BOOL;
END_VAR
//check pumps for errors
bError_PU193 := PU193.bError;
bError_PU393 := PU393.bError;

bError := bError_PU193 OR bError_PU393;
END_METHOD

METHOD PRIVATE LocalControl : BOOL
VAR_INPUT
END_VAR

VAR
	TwoPointControllerOutput : BOOL;
	fSetpointValue: INT;
END_VAR
CASE nControlMode OF
	0: //100%
	nControlMode_RV193 := 0;	//position mode
	fSetPoint_RV193 := 100; 	//100 is fully opened
	
	nControlMode_RV393 := 0;	//position mode
	fSetPoint_RV393 := 100; 	//100 is fully opened
	
	nControlMode_PU193 := 0;
	//fSetPoint_PU393 := 100;
	
	bSetStatusOn_AHU := TRUE;
	//fSetPoint_AHU := 100;
	
	1: //Hysteresis
	nControlMode_RV193 := 0;	//position mode
	nControlMode_RV393 := 0;	//position mode
	nControlMode_PU193 := 0;
	nControlMode_PU393 := 0;
	//fSetPoint_PU393 := 100;
	//fSetPoint_PU193 := 100;
	//fSetPoint_AHU := 100;
	
	TwoPointControllerParameters.tCtrlCycleTime := T#1S;
	TwoPointControllerParameters.tTaskCycleTime := T#10MS;
	IF fHysteresisRange < 1 THEN
		TwoPointControllerParameters.fHysteresisRange := 1;
	ELSE
		TwoPointControllerParameters.fHysteresisRange := fHysteresisRange;
	END_IF;
	
	TwoPointControllerHeating(
			fSetpointValue := fSetPoint,
			fActualValue := stAmbientState.fRoomTemperature,
			bManSyncValue := 0,
			bSync := FALSE,
			emode := 2,
			stParams := TwoPointControllerParameters);
			
	TwoPointControllerCooling(
			fSetpointValue := stAmbientState.fRoomTemperature,
			fActualValue := fSetPoint,
			bManSyncValue := 0,
			bSync := FALSE,
			emode := 2,
			stParams := TwoPointControllerParameters);

	
	IF bHeatingMode THEN
		IF TwoPointControllerHeating.bOut THEN
			fSetPoint_RV393 := 100; 	//100 is fully opened
			bSetStatusOn_PU393 := TRUE;
			bSetStatusOn_AHU := TRUE;
		ELSE
			fSetPoint_RV393 := 0; 	//100 is fully opened
			bSetStatusOn_PU393 := FALSE;
			bSetStatusOn_AHU := FALSE;
		END_IF
	ELSE //cooling mode
		IF TwoPointControllerCooling.bOut THEN
			fSetPoint_RV193 := 100; 	//100 is fully opened
			bSetStatusOn_PU193 := TRUE;
			bSetStatusOn_AHU := TRUE;
		ELSE
			fSetPoint_RV193 := 0; 	//100 is fully opened
			bSetStatusOn_PU193 := FALSE;
			bSetStatusOn_AHU := FALSE;
		END_IF
	END_IF	
	
			
	2: //Continous with PI-Controller
	bSetStatusOn_AHU := TRUE;
	
	nControlMode_PU193 := 0;
	nControlMode_PU393 := 0;
		
	IF bHeatingMode THEN
		nControlMode_RV393 := 1;	//heating mode
		fSetPoint_RV393 := fSetPoint;
		
		bSetStatusOn_PU393 := TRUE;
		bSetStatusOn_PU193 := FALSE;
		
		nControlMode_RV193 := 0;	//turn off other valve
		fSetPoint_RV193 := 0;
	ELSE
		nControlMode_RV193 := 2;	//cooling mode
		fSetPoint_RV193 := fSetPoint;
		
		bSetStatusOn_PU193 := TRUE;
		bSetStatusOn_PU393 := FALSE;
		
		nControlMode_RV393 := 0;	//turn off other valve
		fSetPoint_RV393 := 0;
	END_IF		

END_CASE
END_METHOD

METHOD PROTECTED  Operational : BOOL
VAR_INPUT
END_VAR
VAR_OUTPUT
	bSwitchToWorking : BOOL := FALSE;
END_VAR
IF PU193.bStatusOn OR PU393.bStatusOn THEN
	bSetStatusOn_AHU := TRUE;	
	bSwitchToWorking := TRUE;
END_IF
END_METHOD

METHOD PROTECTED  RampDown : BOOL
VAR_INPUT
END_VAR
VAR_OUTPUT
	bRampDownFinished : BOOL := FALSE;
END_VAR
bSetStatusOn_PU193 := FALSE;
bSetStatusOn_PU393 := FALSE;

bSetStatusOn_AHU := FALSE;

IF NOT PU193.bStatusOn AND NOT PU393.bStatusOn THEN
	bSetStatusOn_RV193 := FALSE;
	bSetStatusOn_RV393 := FALSE;
	
	bStartTimer := TRUE;
	IF Timer.Q THEN
		bRampDownFinished := TRUE;
		bStartTimer := FALSE;
	END_IF
END_IF
END_METHOD

METHOD PROTECTED  RampUp : BOOL
VAR_INPUT
END_VAR
VAR_OUTPUT
	bRampUpFinished : BOOL := FALSE;
END_VAR
IF bHeatingMode THEN
	bSetStatusOn_RV393 := TRUE;
	bSetStatusOn_PU393 := TRUE;
	
	bSetStatusOn_RV193 := FALSE;
	bSetStatusOn_PU193 := FALSE;

ELSE
	bSetStatusOn_RV393 := FALSE;
	bSetStatusOn_PU393 := FALSE;
	
	bSetStatusOn_RV193 := TRUE;
	bSetStatusOn_PU193 := TRUE;
	
END_IF

bRampUpFinished := TRUE;
END_METHOD

METHOD PRIVATE SelectLocalControlMode : BOOL
VAR_INPUT
END_VAR
VAR
END_VAR
IF control.bManualModeActivated THEN
	bHeatingMode := localSetParameters.bHeatingModeManual;
	nControlMode := localSetParameters.nControlModeManual;
	fHysteresisRange := localSetParameters.fHysteresisRangeManual;
ELSIF control.bAlgorithmModeActivated AND bAlgorithmPermission THEN
	bHeatingMode := localSetParameters.bHeatingModeAlgorithm;
	nControlMode := localSetParameters.nControlModeAlgorithm;
	fHysteresisRange := localSetParameters.fHysteresisRangeAlgorithm;
ELSE
	bHeatingMode := bHeatingModeAutomatic;
	nControlMode := nControlModeAutomatic;
	fHysteresisRange := fHysteresisRangeAutomatic;
END_IF
END_METHOD

METHOD PROTECTED   SetSetPointLimits : BOOL
VAR_INPUT
END_VAR
VAR_OUTPUT
END_VAR
aSetPointLimits[1] := localDefaultParameters.aSetPointLimitsTemperature[1];
aSetPointLimits[2] := localDefaultParameters.aSetPointLimitsTemperature[2];
END_METHOD

METHOD PROTECTED  SetState : BOOL
VAR_INPUT
END_VAR
VAR_OUTPUT
END_VAR
fOperatingPoint := stAmbientState.fRoomTemperature;

controlState.bStatusOn := bSetStatusOn;
setPointState.aSetPointLimits := aSetPointLimits;
setPointState.fSetPoint := fSetPoint;
setPointState.fOperatingPoint := fOperatingPoint;
setPointState.sSetPointUnit := 'degreeC';
setPointState.sOperatingPointUnit := 'degreeC';
END_METHOD

METHOD PRIVATE SwitchMode : BOOL
VAR_INPUT
	bSwitchToHeating : BOOL; //if false switch to cooling
END_VAR
VAR_OUTPUT
	bFinishedSwitchMode : BOOL := FALSE;
END_VAR
VAR_INST
	bRampDownFinished : BOOL := FALSE;
END_VAR
IF bSwitchToHeating THEN
	//turn off pump first		
	bSetStatusOn_PU193 := FALSE;
	
	//SV can switch simultanously
	bSetStatusOn_RV193 := FALSE;
	bSetStatusOn_RV393 := TRUE;
	
	bFinishedSwitchMode := FALSE;
	bStartTimer := TRUE;
	IF Timer.Q THEN
		bStartTimer := FALSE;
		bRampDownFinished := TRUE;
		bFinishedSwitchMode := TRUE;
		bSetStatusOn_PU393 := TRUE;
	END_IF
ELSE
	//turn off pumps first		
	bSetStatusOn_PU393 := FALSE;

	//SV can switch simultanously
	bSetStatusOn_RV193 := TRUE;
	bSetStatusOn_RV393 := FALSE;

	bFinishedSwitchMode := FALSE;
	bStartTimer := TRUE;
	IF Timer.Q THEN
		bStartTimer := FALSE;
		bRampDownFinished := TRUE;
		bFinishedSwitchMode := TRUE;
		bSetStatusOn_PU193 := TRUE;
	END_IF
END_IF
END_METHOD

METHOD PROTECTED  Working : BOOL
VAR_INPUT
END_VAR
VAR_OUTPUT
	bSwitchToOperational : BOOL := FALSE;
END_VAR
LocalControl();

IF ((SwitchToHeating.Q OR SwitchToCooling.Q) OR NOT bFinishedSwitchMode) THEN
	
	SwitchMode(bSwitchToHeating := bHeatingMode,
		bFinishedSwitchMode => bFinishedSwitchMode);
END_IF;
END_METHOD

END_FUNCTION_BLOCK

// ---- POUs/01 Actuators/FB_AirHandlingUnit.TcPOU
FUNCTION_BLOCK FB_AirHandlingUnit EXTENDS FB_ActuatorContinous
VAR_INPUT
END_VAR
VAR_OUTPUT
END_VAR
VAR

	localDefaultParameters : ST_AirHandlingUnitDefaultParameters;
	
	//analog converters
	OutputConverter : FB_AnalogOutput(fUpperLimit := 100, fLowerLimit := 0);
	
	//I/O Links
	bSetStatusOn_OUT	AT %Q* : BOOL;
	nSetPoint_OUT 		AT %Q* : INT;
	
END_VAR

MAIN();
OutputConverter(fValue := fSetPoint);

METHOD GetState : BOOL
VAR_INPUT
END_VAR
//local state
bStatusOn := controlState.bStatusOn;
END_METHOD

METHOD PROTECTED  SetSetPointLimits : BOOL
VAR_INPUT
END_VAR
aSetPointLimits[1] := 0;
aSetPointLimits[2] := 100;
END_METHOD

METHOD SetState : BOOL
VAR_INPUT
END_VAR
setPointState.fSetPoint := fSetPoint;
setPointState.aSetPointLimits := aSetPointLimits;
setPointState.sSetPointUnit := 'degreeC';

nSetPoint_OUT := OutputConverter.nValue;  //converts real setpoint for terminal
bSetStatusOn_OUT := NOT bSetStatusOn;		// must be inverted, because AHU is on, when do is 0
END_METHOD

END_FUNCTION_BLOCK

// ---- POUs/04 Systems/FB_CNSystem.TcPOU
FUNCTION_BLOCK FB_CNSystem EXTENDS FB_SystemContinous
VAR_INPUT
END_VAR
VAR_OUTPUT
END_VAR
VAR
	//pumps
	stPU196DefaultParameters : ST_PumpGrundfosMagna3DefaultParameters;
	PU196 : FB_PumpGrundfosMagna3 := (ST_DefaultParameters := stPU196DefaultParameters);
	
	//valves
	stSV196DefaultParameters : ST_DiscreteValveDefaultParameters;
	stSV197DefaultParameters : ST_DiscreteValveDefaultParameters;
	
	SV196 : FB_DiscreteValve := (ST_DefaultParameters := stSV196DefaultParameters);
	SV197 : FB_DiscreteValve := (ST_DefaultParameters := stSV197DefaultParameters);
	
	//sensors
	TVL196 : AutomationBaseClasses.FB_TemperatureSensor; //supply temperature cooling
	TRL196 : AutomationBaseClasses.FB_TemperatureSensor; //return temperature cooling
	
	WMZ196 : FB_MollineC3HeatCounter; //cooling network
	
	//internal variables
	bSetStatusOn_PU196 : BOOL;
	bSetStatusOn_SV196 : BOOL;
	bSetStatusOn_SV197 : BOOL;
	
	//clock
	bStartTimer : BOOL;
	Timer : TON;
	
END_VAR

Timer(IN := bStartTimer,
	PT := T#120S);
MAIN();

//pumps
PU196.GetState_Profibus();
PU196(bSetStatusOnAutomatic := bSetStatusOn_PU196,
	bAlgorithmPermission := bAlgorithmPermission,
	fSetPointAutomatic := fSetPoint,
	nControlModeAutomatic := 0);
PU196.SetState_Profibus();

//valves
SV196.GetState_BI();
SV196(bSetStatusOnAutomatic := bSetStatusOn_SV196,
	bAlgorithmPermission := bAlgorithmPermission);
SV196.SetState_BO();

SV197.GetState_BI();
SV197(bSetStatusOnAutomatic := bSetStatusOn_SV197,
	bAlgorithmPermission := bAlgorithmPermission);
SV197.SetState_BO();

//sensors
TVL196();
TVL196.GetState_AI();
TRL196();
TRL196.GetState_AI();

WMZ196(aHeatCounterTelegramm := MBus.Telegramm_WMZ_196);

METHOD PROTECTED  CheckError : BOOL
VAR_INPUT
END_VAR
VAR_OUTPUT
	bError : BOOL;
END_VAR
VAR
	bError_PU196 : BOOL;
END_VAR
bError := PU196.bError;
END_METHOD

METHOD PROTECTED  Operational : BOOL
VAR_INPUT
END_VAR
VAR_OUTPUT
	bSwitchToWorking : BOOL := FALSE;
END_VAR
bSetStatusOn_PU196 := TRUE;

IF PU196.bStatusOn THEN
	bSwitchToWorking := TRUE;
END_IF
END_METHOD

METHOD PROTECTED  RampDown : BOOL
VAR_INPUT
END_VAR
VAR_OUTPUT
	bRampDownFinished : BOOL := FALSE;
END_VAR
bSetStatusOn_PU196 := FALSE;

IF NOT PU196.bStatusOn THEN
	bSetStatusOn_SV196 := FALSE;
	bSetStatusOn_SV197 := FALSE;
	
	bStartTimer := TRUE;
	IF Timer.Q THEN
		bRampDownFinished := TRUE;
		bStartTimer := FALSE;
	END_IF
END_IF
END_METHOD

METHOD PROTECTED  RampUp : BOOL
VAR_INPUT
END_VAR
VAR_OUTPUT
	bRampUpFinished : BOOL := FALSE;
END_VAR
bSetStatusOn_SV196 := TRUE;
bSetStatusOn_SV197 := TRUE;

bStartTimer := TRUE;
IF Timer.Q THEN
	bStartTimer := FALSE;
	bRampUpFinished := TRUE;
END_IF
END_METHOD

METHOD PROTECTED   SetSetPointLimits : BOOL
VAR_INPUT
END_VAR
VAR_OUTPUT
END_VAR
aSetPointLimits[1] := 0;
aSetPointLimits[2] := 100;
END_METHOD

METHOD PROTECTED  SetState : BOOL
VAR_INPUT
END_VAR
VAR_OUTPUT
END_VAR
controlState.bStatusOn := bSetStatusOn;
setPointState.aSetPointLimits := aSetPointLimits;
setPointState.fSetPoint := fSetPoint;
setPointState.fOperatingPoint := fOperatingPoint;
setPointState.sSetPointUnit := 'percent';
setPointState.sOperatingPointUnit := 'percent';
END_METHOD

METHOD PROTECTED  Working : BOOL
VAR_INPUT
END_VAR
VAR_OUTPUT
	bSwitchToOperational : BOOL := FALSE;
END_VAR
//empty
END_METHOD

END_FUNCTION_BLOCK

// ---- POUs/04 Systems/FB_HNLTSystem.TcPOU
FUNCTION_BLOCK FB_HNLTSystem
VAR_INPUT
END_VAR
VAR_OUTPUT
END_VAR
VAR
	
	// heat counters
	WMZ246 : FB_MollineC3HeatCounter;
	WMZ247 : FB_MollineC3HeatCounter;

END_VAR

WMZ246(aHeatCounterTelegramm := MBus.Telegramm_WMZ_246);
WMZ247(aHeatCounterTelegramm := MBus.Telegramm_WMZ_247);

END_FUNCTION_BLOCK

// ---- POUs/04 Systems/FB_PowerControlledHeaterSystem.TcPOU
FUNCTION_BLOCK FB_PowerControlledHeaterSystem EXTENDS FB_SystemContinous
VAR_INPUT
END_VAR
VAR_OUTPUT
END_VAR
VAR
	
	localDefaultParameters : ST_PowerControlledHeaterDefaultParameters;
	{attribute 'OPC.UA.DA' := '1'}	
	localState : ST_PowerControlledHeaterState;
	
	//system components
	fan 			: FB_PowerControlledHeaterFan;
	contactor1 		: FB_PowerControlledHeaterContactor;
	contactor2 		: FB_PowerControlledHeaterContactor;
	thyristor1 		: FB_PowerControlledHeaterThyristor;
	thyristor2 		: FB_PowerControlledHeaterThyristor;

	//internal variables
	bSetStatusOn_fan : BOOL;
	bSetStatusOn_contactors : BOOL;
	bSetStatusOn_thyristors : BOOL;
	
	fPowerTotal : REAL;
	fTemperatureMax : REAL;

	//sensors
	THeater1 : FB_TemperatureSensorPCH;
	THeater2 : FB_TemperatureSensorPCH;
	THeater3 : FB_TemperatureSensorPCH;
	THeater4 : FB_TemperatureSensorPCH;

	PowerPhase1 : FB_JanitzaSensor;
	PowerPhase2 : FB_JanitzaSensor;
	PowerPhase3 : FB_JanitzaSensor;
	
END_VAR

MAIN();

fan(bSetStatusOnAutomatic := bSetStatusOn_fan,
	bAlgorithmPermission := bAlgorithmPermission);
fan.SetState_BO();

contactor1(bSetStatusOnAutomatic := bSetStatusOn_contactors,
	bAlgorithmPermission := bAlgorithmPermission);
contactor1.SetState_BO();

contactor2(bSetStatusOnAutomatic := bSetStatusOn_contactors,
	bAlgorithmPermission := bAlgorithmPermission);
contactor2.SetState_BO();	

//sensors
THeater1();
THeater1.GetState_AI();
THeater2();
THeater2.GetState_AI();
THeater3();
THeater3.GetState_AI();
THeater4();
THeater4.GetState_AI();

PowerPhase1();
PowerPhase1.GetState_AI();
PowerPhase2();
PowerPhase2.GetState_AI();
PowerPhase3();
PowerPhase3.GetState_AI();

fPowerTotal := PowerPhase1.fPower + PowerPhase2.fPower + PowerPhase3.fPower; //calculate total power
fTemperatureMax := MAX(THeater1.fTemperature, THeater2.fTemperature, THeater3.fTemperature, THeater4.fTemperature); //find max temperatur for temperature permission

thyristor1(bSetStatusOnAutomatic := bSetStatusOn_thyristors,
	bAlgorithmPermission := bAlgorithmPermission,
	fSetPointAutomatic := fSetPoint,
	fPowerTotal := fPowerTotal,
	fTemperature := fTemperatureMax);
thyristor1.SetState();
	
thyristor2(bSetStatusOnAutomatic := bSetStatusOn_thyristors,
	bAlgorithmPermission := bAlgorithmPermission,
	fSetPointAutomatic := fSetPoint,
	fPowerTotal := fPowerTotal,
	fTemperature := fTemperatureMax);	
thyristor2.SetState();

METHOD PROTECTED  CheckError : BOOL
VAR_INPUT
END_VAR
VAR_OUTPUT
	bError : BOOL;
END_VAR
VAR
END_VAR
//check for temperature permission of thyristors
bError := thyristor1.bError OR thyristor2.bError;
END_METHOD

METHOD PROTECTED  Operational : BOOL
VAR_INPUT
END_VAR
VAR_OUTPUT
	bSwitchToWorking : BOOL := FALSE;
END_VAR
bSetStatusOn_thyristors := TRUE;
bSwitchToWorking := TRUE;
END_METHOD

METHOD PROTECTED  RampDown : BOOL
VAR_INPUT
END_VAR
VAR_OUTPUT
	bRampDownFinished : BOOL := FALSE;
END_VAR
bSetStatusOn_fan := FALSE;
bSetStatusOn_thyristors := FALSE;

//prevent switching contactors if total power is too high
IF fPowerTotal < 50 THEN
	bSetStatusOn_contactors := FALSE;
	bRampDownFinished := TRUE;
END_IF
END_METHOD

METHOD PROTECTED  RampUp : BOOL
VAR_INPUT
END_VAR
VAR_OUTPUT
	bRampUpFinished : BOOL := FALSE;
END_VAR
bSetStatusOn_fan := TRUE;
bSetStatusOn_contactors := TRUE;

bRampUpFinished := TRUE;
END_METHOD

METHOD PROTECTED   SetSetPointLimits : BOOL
VAR_INPUT
END_VAR
VAR_OUTPUT
END_VAR
aSetPointLimits[1] := 0;
aSetPointLimits[2] := 5000;
END_METHOD

METHOD PROTECTED  SetState : BOOL
VAR_INPUT
END_VAR
VAR_OUTPUT
END_VAR
controlState.bStatusOn := bSetStatusOn;
setPointState.aSetPointLimits := aSetPointLimits;
setPointState.fSetPoint := fSetPoint;
setPointState.fOperatingPoint := fPowerTotal;
setPointState.sSetPointUnit := 'W';
setPointState.sOperatingPointUnit := 'W';
localState.fPowerTotal := fPowerTotal;
END_METHOD

METHOD PROTECTED  Working : BOOL
VAR_INPUT
END_VAR
VAR_OUTPUT
	bSwitchToOperational : BOOL := FALSE;
END_VAR
//empty
END_METHOD

END_FUNCTION_BLOCK

// ---- POUs/01 Actuators/FB_PowerControlledHeaterFan.TcPOU
FUNCTION_BLOCK FB_PowerControlledHeaterFan EXTENDS FB_Actuator2Point

VAR
	
	//I/O Links	
	bSetStatusOn_OUT 	AT %Q*	: 	BOOL := FALSE;		
	
END_VAR

SelectControlMode();

METHOD SetState_BO : BOOL
VAR_INPUT
END_VAR
//output
bSetStatusOn_OUT := bSetStatusOn;
END_METHOD

END_FUNCTION_BLOCK

// ---- POUs/01 Actuators/FB_PowerControlledHeaterContactor.TcPOU
FUNCTION_BLOCK FB_PowerControlledHeaterContactor EXTENDS FB_Actuator2Point

VAR
	
	//I/O Links	
	bSetStatusOn_OUT 	AT %Q*	: 	BOOL := FALSE;		
	
END_VAR

SelectControlMode();

METHOD SetState_BO : BOOL
VAR_INPUT
END_VAR
//output
bSetStatusOn_OUT := bSetStatusOn;
END_METHOD

END_FUNCTION_BLOCK

// ---- POUs/01 Actuators/FB_PowerControlledHeaterThyristor.TcPOU
FUNCTION_BLOCK FB_PowerControlledHeaterThyristor EXTENDS FB_ActuatorContinous
VAR_INPUT
	fPowerTotal : REAL;
	fTemperature : REAL;
END_VAR
VAR
	stTemperatureCheckDefaultParameters : ST_RangeCheckDefaultParameters := (tTaskCycleTime := GlobalVariables.tCtrlCycleTime_MAIN, tCtrlCycleTime := GlobalVariables.tCtrlCycleTime_MAIN, fRestoreDifference := 10);
	Temperature_Check : FB_RangeCheck := (ST_DefaultParameters := stTemperatureCheckDefaultParameters);
	
	//controller
	PID_Controller				: FB_CTRL_PID;
	PID_Controller_Parameters	: ST_CTRL_PID_PARAMS;
	
	fSetPoint_internal 			: REAL; //internal setpoint between 0 and 32767
	bTemperaturePermission		: BOOL;
	
	//I/O Links
	nSetPoint_OUT 		AT %Q* : INT;	
	
END_VAR
VAR_OUTPUT
	bError 						: BOOL;
	
END_VAR

Temperature_Check(fInput := fTemperature,
	fLowerLimit := -99,
	fUpperLimit := 100);
bTemperaturePermission := Temperature_Check.bPermission;
	
MAIN();
LocalControl();

METHOD GetState : BOOL
VAR_INPUT
END_VAR
//local state
bStatusOn := controlState.bStatusOn;
END_METHOD

METHOD LocalControl : BOOL
VAR_INPUT
END_VAR
PID_Controller_Parameters.fKp:=1.8;
PID_Controller_Parameters.tTn:= T#1600MS;
PID_Controller_Parameters.tTv:=T#4MS;
PID_Controller_Parameters.fOutMaxLimit:= 32767;
PID_Controller_Parameters.fOutMinLimit:=  0;
PID_Controller_Parameters.tCtrlCycleTime:= T#5S;
PID_Controller_Parameters.tTaskCycleTime:= T#10MS;
PID_Controller_Parameters.bARWOnIPartOnly:= FALSE; 

PID_Controller(fSetpointValue:=fSetPoint, 
fActualValue:=fPowerTotal, 
fManSyncValue:=0, 
bSync:=FALSE, 
eMode:=2, 
bHold:=FALSE, 
stParams:=PID_Controller_Parameters);

//overwrite internal setpoint, if Temperatur is too high
IF bSetStatusOn AND bTemperaturePermission THEN
	fSetPoint_internal := LREAL_TO_REAL(PID_Controller.fOut);
	bError := FALSE;
ELSE
	fSetPoint_internal := 0;
	bError := TRUE;
END_IF
END_METHOD

METHOD PROTECTED  SetSetPointLimits : BOOL
VAR_INPUT
END_VAR
aSetPointLimits[1] := 0;
aSetPointLimits[2] := 5000;
END_METHOD

METHOD SetState : BOOL
VAR_INPUT
END_VAR
setPointState.fSetPoint := fSetPoint_internal;
setPointState.aSetPointLimits := aSetPointLimits;
setPointState.sSetPointUnit := 'W';

nSetPoint_OUT := REAL_TO_INT(fSetPoint_internal);
END_METHOD

END_FUNCTION_BLOCK

// ---- POUs/02 Sensors/FB_TemperatureSensorPCH.TcPOU
FUNCTION_BLOCK FB_TemperatureSensorPCH EXTENDS FB_Sensor
VAR_INPUT
END_VAR
VAR_OUTPUT
	fTemperature : REAL; //measured temperature in °C
END_VAR
VAR
	//I/O-Links
	temperature_IN AT %I* : INT;
	
END_VAR

METHOD GetState_AI : BOOL
VAR_INPUT
END_VAR
fTemperature := temperature_IN*0.1; //conversion

//sensor state
sensorState.fValue := fTemperature;
sensorState.sUnit := 'degreeC';
END_METHOD

END_FUNCTION_BLOCK

// ---- POUs/02 Sensors/FB_JanitzaSensor.TcPOU
FUNCTION_BLOCK FB_JanitzaSensor EXTENDS FB_Sensor
VAR_INPUT
END_VAR
VAR_OUTPUT
	fPower : REAL; //measured power in watt
END_VAR
VAR
	//I/O-Links
	power_IN AT %I* : REAL;
	
END_VAR

METHOD GetState_AI : BOOL
VAR_INPUT
END_VAR
fPower := power_IN;

//sensor state
sensorState.fValue := fPower;
sensorState.sUnit := 'Watt';
END_METHOD

END_FUNCTION_BLOCK
